FUNCTION_BLOCK SubscribeEvent (* Subscribe Event Function Block *)
  (* Standard: 61499-2; Description: Copyright (c) 2019 fortiss GmbH This program and the accompanying materials are made available under the terms of the Eclipse Public License 2.0 which is available at https://www.eclipse.org/legal/epl-2.0/ SPDX-License-Identifier: EPL-2.0 *)
  (* Version 1.0, 2019-09-18, Cabral, fortiss GmbH *)
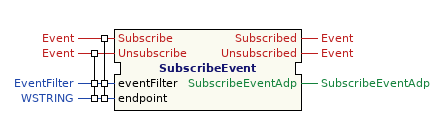
  EVENT_INPUT
    Subscribe WITH eventFilter, endpoint; (* Initialization Request *)
    Unsubscribe WITH eventFilter, endpoint; (* Normal Execution Request *)
  END_EVENT
  EVENT_OUTPUT
    Subscribed; (* Subscribe finished *)
    Unsubscribed; (* Unsubscribe from event *)
  END_EVENT
  VAR_INPUT
    eventFilter : EventFilter; (* Event filter *)
    endpoint : WSTRING; (* Endpoint (IP:PORT/URI) of the Service Registry (not officially in the documentation, but it simplifies the FBs) *)
  END_VAR
  PLUGS
    SubscribeEventAdp : SubscribeEventAdp; (* Subscribe event adapter *)
  END_PLUGS
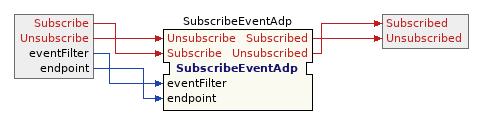
  EVENT_CONNECTIONS
    Unsubscribe TO SubscribeEventAdp.Unsubscribe;
    Subscribe TO SubscribeEventAdp.Subscribe;
    SubscribeEventAdp.Subscribed TO Subscribed;
    SubscribeEventAdp.Unsubscribed TO Unsubscribed;
  END_CONNECTIONS
  DATA_CONNECTIONS
    eventFilter TO SubscribeEventAdp.eventFilter;
    endpoint TO SubscribeEventAdp.endpoint;
  END_CONNECTIONS
END_FUNCTION_BLOCK
